Staubli VAL3: start.pgx

program start()
  local num l_nRound
  local num l_nDieEyes
  local bool l_bPlayer1Plays
  local num l_nAdd
  local num l_nElement
  local num l_nCoord
  local num l_nRange
  local num l_nCommand
  local num l_nRangeX
  local num l_nRangeZ
  local num l_nRangeY
  local bool l_bInRange
begin

  call util:readFile("input_day22.txt",  sInput)
  // sInput[0] = "on x=10..12,y=10..12,z=10..12"

  call str:splitString(sInput," ", lResult)

  resize(bGrid,1,101)
  resize(bGrid,2,101)
  resize(bGrid,3,101)

  resize(sCommand,1,size(lResult))
  for l_nElement = 0 to size(lResult)-1
    ? l_nElement
    sCommand[l_nElement] = lResult[l_nElement].sString[0]
    call str:splitString(lResult[l_nElement].sString[1], ",", lResultCoord)

    call str:replacePattern(lResultCoord.sString[0],"x=", "", sCoord_X)
    call str:replacePattern(lResultCoord.sString[1],"y=", "", sCoord_Y)
    call str:replacePattern(lResultCoord.sString[2],"z=", "", sCoord_Z)

    resize(sCoord_X,1,1)
    resize(sCoord_Y,1,1)
    resize(sCoord_Z,1,1)

    // get coordinates as number
    call str:splitString(sCoord_X, "..", lResultCoord)
    call util:vec2num(lResultCoord.sString, nCoord_X)

    if nCoord_X[0] >= -50 and nCoord_X[1]<= 50
      l_bInRange = true
      call util:range(nCoord_X[0]+50, nCoord_X[1]+1+50, 1, nRangeX)
    else
      l_bInRange = false
    endIf

    if l_bInRange
      call str:splitString(sCoord_Y, "..", lResultCoord)
      call util:vec2num(lResultCoord.sString, nCoord_Y)
      if nCoord_Y[0] >= -50 and nCoord_Y[1]<= 50
        l_bInRange = true
        call util:range(nCoord_Y[0]+50, nCoord_Y[1]+1+50, 1, nRangeY)
      else
        l_bInRange = false
      endIf
    endIf

    if l_bInRange
      call str:splitString(sCoord_Z, "..", lResultCoord)
      call util:vec2num(lResultCoord.sString, nCoord_Z)
      if nCoord_Z[0] >= -50 and nCoord_Z[1]<= 50
        l_bInRange = true
        call util:range(nCoord_Z[0]+50, nCoord_Z[1]+1+50, 1, nRangeZ)
      else
        l_bInRange = false
      endIf
    endIf

    if l_bInRange
      // fill 3d-matrix
      for l_nRangeX = 0 to size(nRangeX)-1
        for l_nRangeY = 0 to size(nRangeY)-1
          for l_nRangeZ = 0 to size(nRangeZ)-1
            if sCommand[l_nElement] == "on"
              bGrid[nRangeX[l_nRangeX], nRangeY[l_nRangeY], nRangeZ[l_nRangeZ]] = true
            else
              bGrid[nRangeX[l_nRangeX], nRangeY[l_nRangeY], nRangeZ[l_nRangeZ]] = false
            endIf
          endFor
        endFor
      endFor
    endIf

  endFor

  // count TRUEs
  call util:countBool3D(bGrid, nResult)
  call util:printNum(nResult)
  // 603661

end
